FUNCTION_BLOCK ExerciseFireBypassDamperParameters
VAR_INPUT
	TimeChannel: TimeChannelSettings;
	StartManualExercise: BOOL;
	ExerciseStatus: BOOL;
	CloseFTXDamper: BOOL;
	StopSystem: BOOL;
END_VAR
VAR_OUTPUT
END_VAR
VAR
END_VAR

END_FUNCTION_BLOCK

(* stored: Version 1.1.0.1, ProductVersion 3.1.4024.6
   POU ExerciseFireBypassDamperParameters: Id {cd9de177-1e8e-4f3c-a828-db1036ea21fb}, SpecialFunc None *)
